FUNCTION_BLOCK Disc_brake
VAR_INPUT
	S1:REAL; (*Raw analogue value from proxmity transducer in brake caliper module 1*)
	S2:REAL; (*Raw analogue value from proxmity transducer in brake caliper module 2*)
	Pressure:BOOL; (*This input must be active when the pressure is above the threshold used for broken spring detection*)
	Raw_min:REAL; (*Minimum value of raw sensor analogue inputs*)
	Raw_max:REAL; (*Maximum value of raw sensor analogue inputs*)
	Pos_min:REAL; (*Position value corresponding to minimum raw value (typically in mm)*)
	Pos_max:REAL; (*Position value corresponding to maximum raw value (typically in mm)*)
	mA_min:REAL; (*Milliamp value corresponding to minimum raw value (typically 3 to 4mA for 4-20mA transducers)*)
	mA_max:REAL; (*Milliamp value corresponding to maximum raw value (typically 20mA for 4-20mA transducers)*)
	Range_min:REAL; (*Minimum allowed raw value. A lower value will result in an out of range error.*)
	Range_max:REAL; (*Maximum allowed raw value. A lower value will result in an out of range error*)
	Broken_wire:REAL; (*Raw value below which a 4-20mA transducer can be considered open circuit*)
	Off_pos:REAL; (*Position (scaled) value below which the brake module can be considered to be in the "off" position*)
	Rubbing_pos:REAL; (*Position (scaled) value above which the brake module can be considered to be rubbing*)
	On_pos:REAL; (*Average position (scaled) value above which the brake modules can be considered to be "on"*)
	Wear_pos:REAL; (*Average position (scaled) value above which the brake pads can be considered to be "worn"*)
	Speed:REAL;
	Brake_rubbing_speed:REAL;
	Brake_rubbing_on_delay:TIME;
	Colour_scheme:INT; (*An integer value corresponding to the analogue colour scheme to be used on the HMI*)
END_VAR
VAR_OUTPUT
	Pos1:REAL; (*Scaled position value for sensor 1 (typically in mm)*)
	Pos2:REAL; (*Scaled position value for sensor 2 (typically in mm)*)
	mA1:REAL; (*Milliamp value for sensor 1 (for 4-20mA transducers)*)
	mA2:REAL; (*Milliamp value for sensor 2 (for 4-20mA transducers)*)
	Off:BOOL; (*Both brake modules in the "off" position*)
	Rubbing:BOOL; (*At least one of the brake modules is past the "rubbing" position*)
	Brake_on:BOOL; (*The average value of the modules positions is greater than the "on" distance*)
	Wear:BOOL; (*The average value of the modules positions is greater than the "wear" distance*)
	Broken_spring1:BOOL; (*Module 1 has a broken spring (the off position was reached with insufficient pressure)*)
	Broken_spring2:BOOL; (*Module 2 has a broken spring (the off position was reached with insufficient pressure)*)
	S1_out_of_range:BOOL; (*The analogue value of sensor 1 is out of range*)
	S2_out_of_range:BOOL; (*The analogue value of sensor 2 is out of range*)
	S1_broken_wire:BOOL; (*The analogue value of sensor 1 is out of range*)
	S2_broken_wire:BOOL; (*The analogue value of sensor 2 is out of range*)
	tr_Rubbing1:BOOL; (*Side 1 rubbing above allowed speed*)
	tr_Rubbing2:BOOL; (*Side 2 rubbing above allowed speed*)
	HMI1:dut_hmi_Analogue; (*Data structure containing sensor 1 data for HMI*)
	HMI2:dut_hmi_Analogue; (*Data structure containing sensor 2 data for HMI*)
END_VAR
VAR
	Ave_pos:REAL;
	Off1:BOOL;
	Off2:BOOL;
	S1_rubbing:BOOL;
	S2_rubbing:BOOL;
	Raw_to_scaled_0: Raw_to_scaled;
	Raw_to_scaled_1: Raw_to_scaled;
END_VAR

Disc_brake_scaling();
Disc_brake_positions();
Disc_brake_faults();
Disc_brake_HMI();

METHOD Disc_brake_faults
VAR_INPUT
END_VAR
VAR_INST // added by the converter: edge detectors and wires of the graphical bodies
    _w1, _w2, _w3 : BOOL;
END_VAR
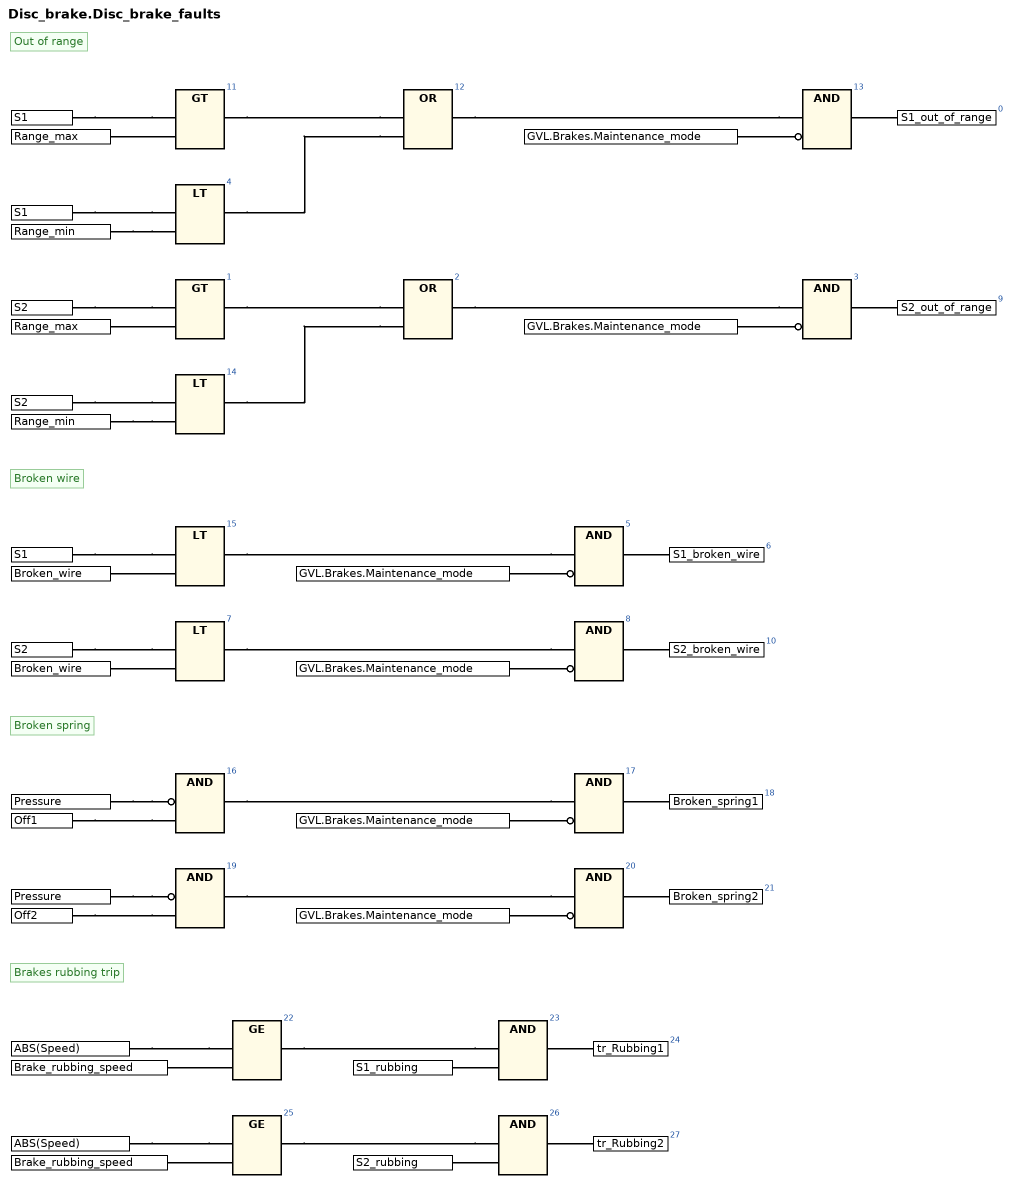
S1_out_of_range := _w1;
S1_broken_wire := _w3 AND NOT GVL.Brakes.Maintenance_mode;
S2_out_of_range := (S2 > Range_max OR _w2) AND NOT GVL.Brakes.Maintenance_mode;
S2_broken_wire := S2 < Broken_wire AND NOT GVL.Brakes.Maintenance_mode;
// Out of range
_w1 := (S1 > Range_max OR S1 < Range_min) AND NOT GVL.Brakes.Maintenance_mode;
_w2 := S2 < Range_min;
// Broken wire
_w3 := S1 < Broken_wire;
// Broken spring
Broken_spring1 := (NOT Pressure AND Off1) AND NOT GVL.Brakes.Maintenance_mode;
Broken_spring2 := (NOT Pressure AND Off2) AND NOT GVL.Brakes.Maintenance_mode;
// Brakes rubbing trip
tr_Rubbing1 := (ABS(Speed)) >= Brake_rubbing_speed AND S1_rubbing;
tr_Rubbing2 := (ABS(Speed)) >= Brake_rubbing_speed AND S2_rubbing;
END_METHOD

METHOD Disc_brake_HMI
VAR_INPUT
END_VAR
VAR_INST // added by the converter: edge detectors and wires of the graphical bodies
    _w1, _w2, _w3, _w4, _w8, _w9, _w10, _w12, _w13, _w14, _w15, _w16, _w17 : ANY;
    _w5 : REAL;
    _w6, _w7, _w11 : BOOL;
END_VAR
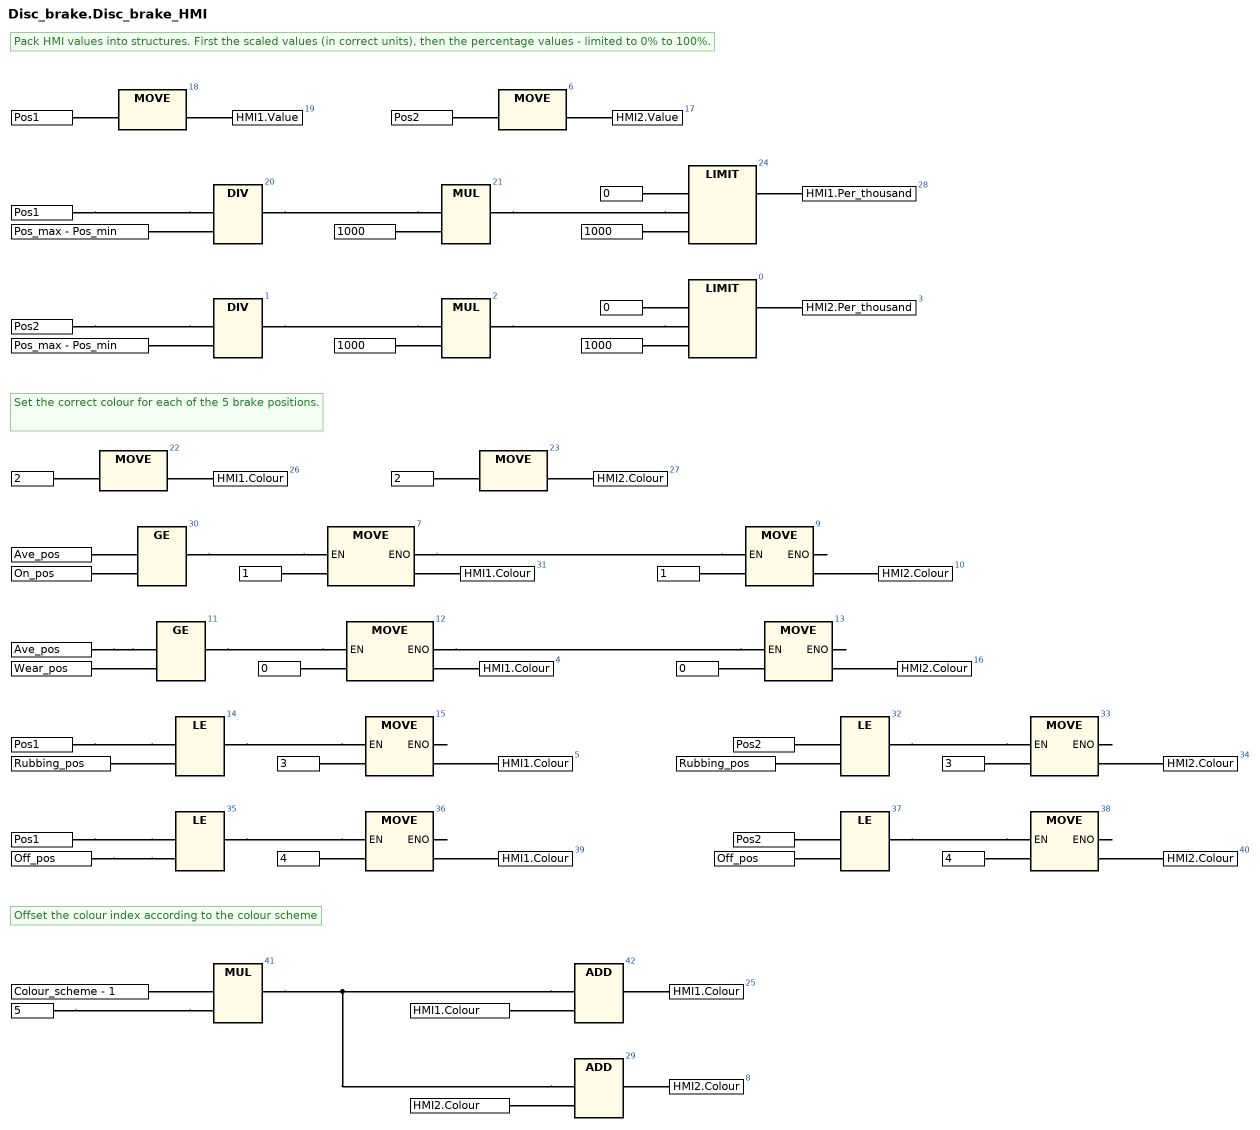
_w2 := LIMIT(0, _w1, 1000);
_w1 := (Pos2 / (Pos_max - Pos_min)) * 1000;
HMI2.Per_thousand := _w2;
HMI1.Colour := _w3;
HMI1.Colour := _w4;
_w5 := Pos2;
_w7 := _w6;
IF _w7 THEN _w8 := 1; END_IF
HMI2.Colour := _w9;
IF _w7 THEN _w10 := 1; END_IF
HMI2.Colour := _w10;
_w11 := Ave_pos >= Wear_pos;
IF _w11 THEN _w3 := 0; END_IF
IF _w11 THEN _w12 := 0; END_IF
IF Pos1 <= Rubbing_pos THEN _w4 := 3; END_IF
HMI2.Colour := _w12;
HMI2.Value := _w5;
// Pack HMI values into structures. First the scaled values (in correct units), then the percentage values - limited to 0% to 100%.
HMI1.Value := Pos1;
// Set the correct colour for each of the 5 brake positions.
HMI1.Colour := _w13;
HMI1.Colour := 2;
HMI2.Colour := 2;
HMI1.Per_thousand := LIMIT(0, (Pos1 / (Pos_max - Pos_min)) * 1000, 1000);
_w9 := _w14 + HMI2.Colour;
_w6 := Ave_pos >= On_pos;
HMI1.Colour := _w8;
IF Pos2 <= Rubbing_pos THEN _w15 := 3; END_IF
HMI2.Colour := _w15;
IF Pos1 <= Off_pos THEN _w16 := 4; END_IF
IF Pos2 <= Off_pos THEN _w17 := 4; END_IF
HMI1.Colour := _w16;
HMI2.Colour := _w17;
// Offset the colour index according to the colour scheme
_w14 := (Colour_scheme - 1) * 5;
_w13 := _w14 + HMI1.Colour;
END_METHOD

METHOD Disc_brake_positions
VAR_INPUT
END_VAR
VAR_INST // added by the converter: edge detectors and wires of the graphical bodies
    _w1, _w2, _w3, _w4, _w5, _w6 : BOOL;
END_VAR
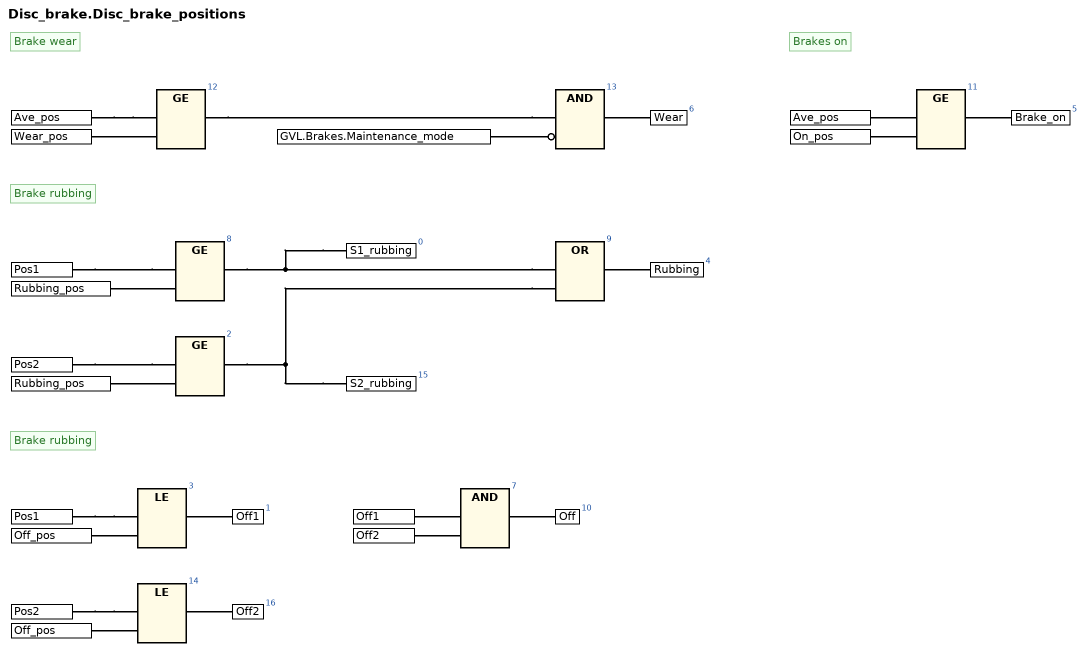
S1_rubbing := _w1;
Off1 := _w2;
_w3 := Pos2 >= Rubbing_pos;
// Brake rubbing
_w2 := Pos1 <= Off_pos;
Rubbing := _w4;
Brake_on := _w5;
Wear := _w6;
// Brake rubbing
_w1 := Pos1 >= Rubbing_pos;
_w4 := _w1 OR _w3;
Off := Off1 AND Off2;
// Brakes on
_w5 := Ave_pos >= On_pos;
// Brake wear
_w6 := Ave_pos >= Wear_pos AND NOT GVL.Brakes.Maintenance_mode;
S2_rubbing := _w3;
Off2 := Pos2 <= Off_pos;
END_METHOD

METHOD Disc_brake_scaling
VAR_INPUT
END_VAR

VAR
END_VAR
VAR_INST // added by the converter: edge detectors and wires of the graphical bodies
    _w1 : REAL;
END_VAR
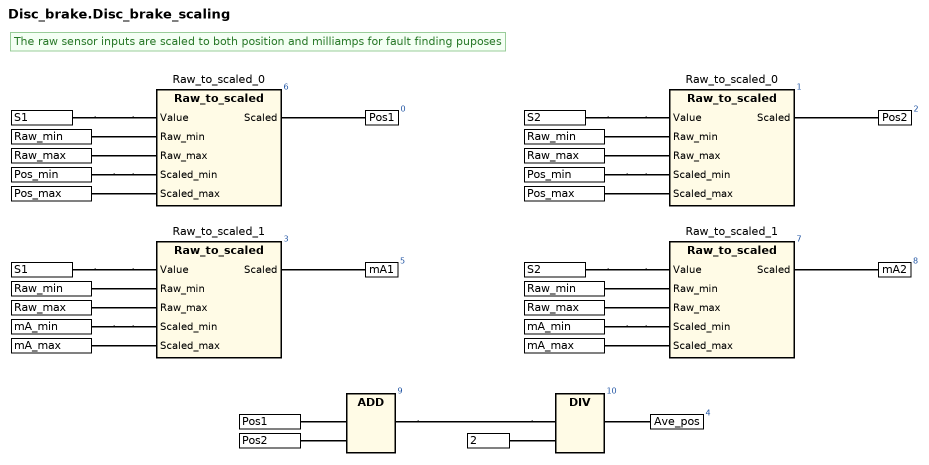
Pos1 := Raw_to_scaled_0.Scaled;
Raw_to_scaled_0(
    Value := S2,
    Raw_min := Raw_min,
    Raw_max := Raw_max,
    Scaled_min := Pos_min,
    Scaled_max := Pos_max); // Raw_to_scaled
Pos2 := Raw_to_scaled_0.Scaled;
Raw_to_scaled_1(
    Value := S1,
    Raw_min := Raw_min,
    Raw_max := Raw_max,
    Scaled_min := mA_min,
    Scaled_max := mA_max); // Raw_to_scaled
Ave_pos := _w1;
mA1 := Raw_to_scaled_1.Scaled;
// The raw sensor inputs are scaled to both position and milliamps for fault finding puposes
Raw_to_scaled_0(
    Value := S1,
    Raw_min := Raw_min,
    Raw_max := Raw_max,
    Scaled_min := Pos_min,
    Scaled_max := Pos_max); // Raw_to_scaled
Raw_to_scaled_1(
    Value := S2,
    Raw_min := Raw_min,
    Raw_max := Raw_max,
    Scaled_min := mA_min,
    Scaled_max := mA_max); // Raw_to_scaled
mA2 := Raw_to_scaled_1.Scaled;
_w1 := (Pos1 + Pos2) / 2;
END_METHOD

END_FUNCTION_BLOCK

(* stored: Version 1.1.0.1, ProductVersion 3.1.4024.0
   POU Disc_brake: Id {979e2970-fb6e-4c17-b656-0f02b5a10666}, SpecialFunc None
   Method Disc_brake_faults: Id {d16c184a-2791-4e01-9656-e3282c0e82ae}
   Method Disc_brake_HMI: Id {6c0f07e7-f527-4038-b75d-f839fd30dc79}
   Method Disc_brake_positions: Id {b372afdc-fe04-4c87-bc80-583b38b62444}
   Method Disc_brake_scaling: Id {e82b97ed-5d4c-4e36-978d-45b8667d8c9b} *)
